// TIA Portal V17 export
// export: Created 2025-03-13T10:31:25.9851877Z, ExportSetting WithDefaults, DisplayName Totally Integrated Automation Portal, DisplayVersion V17 Update 8, DisplayName TIA Portal Openness, DisplayVersion V17 Update 8, DisplayName TIA Portal Version Control Interface, DisplayVersion V17, DisplayName SINAMICS Startdrive Advanced, DisplayVersion V17 SP2, DisplayName SINAMICS Startdrive G110M, G120, G120C, G120D, G120P, G115D, DisplayVersion V17 SP2, DisplayName SINAMICS Startdrive G130, G150, S120, S150, SINAMICS MV, S210, DisplayVersion V17 SP2, DisplayName STEP 7 Professional, DisplayVersion V17 Update 8, DisplayName SINUMERIK ONE STEP 7 Toolbox, DisplayVersion V17 Update 12, DisplayName SINUMERIK 840D sl STEP 7 Toolbox, DisplayVersion V17 Update 12, DisplayName STEP 7 Safety, DisplayVersion V17 Update 6, DisplayName WinCC Advanced, DisplayVersion V17 Update 8
TYPE "FULL_DEPTH_CLADDING"
// stored: IsFailsafeCompliant false
   STRUCT
      FULL_DEPTH : Bool;   // FULL DEPTH / TOTAL FULL DEPTH
      FULL_DEPTH_STA_1 : Bool;   // FULL DEPTH 1 / FULL DEPTH STATION 1
      FULL_DEPTH_STA_2 : Bool;   // FULL DEPTH 2 / FULL DEPTH STATION 2
      FULL_DEPTH_STA_3 : Bool;   // FULL DEPTH 3 / FULL DEPTH STATION 3
      FULL_DEPTH_STA_4 : Bool;   // FULL DEPTH 4 / FULL DEPTH STATION 4
      FULL_DEPTH_STA_5 : Bool;   // FULL DEPTH 5 / FULL DEPTH STATION 5
      FULL_DEPTH_STA_6 : Bool;   // FULL DEPTH 6 / FULL DEPTH STATION 6
      FULL_DEPTH_STA_7 : Bool;   // FULL DEPTH 7 / FULL DEPTH STATION 7
      PART_REJECTED_FIXTURE : Bool;   // PART REJECTED FIXTURE 1 / PART REJECTED FIXTURE
      AUX_FULL_DEPTH_STA_1 : Bool;   // AUXILIARY FULL DEPTH 1 / AUXILIARY FULL DEPTH STATION 1
      AUX_FULL_DEPTH_STA_2 : Bool;   // AUXILIARY FULL DEPTH 2 / AUXILIARY FULL DEPTH STATION 2
      AUX_FULL_DEPTH_STA_3 : Bool;   // AUXILIARY FULL DEPTH 3 / AUXILIARY FULL DEPTH STATION 3
      AUX_FULL_DEPTH_STA_4 : Bool;   // AUXILIARY FULL DEPTH 4 / AUXILIARY FULL DEPTH STATION 4
      AUX_FULL_DEPTH_STA_5 : Bool;   // AUXILIARY FULL DEPTH 5 / AUXILIARY FULL DEPTH STATION 5
      AUX_FULL_DEPTH_STA_6 : Bool;   // AUXILIARY FULL DEPTH 6 / AUXILIARY FULL DEPTH STATION 6
      AUX_FULL_DEPTH_STA_7 : Bool;   // AUXILIARY FULL DEPTH 7 / AUXILIARY FULL DEPTH STATION 7
      AUX_FULL_DEPTH_STA_8 : Bool;   // AUXILIARY FULL DEPTH 8 / AUXILIARY FULL DEPTH STATION 8
      AUX_FULL_DEPTH_PULSE_STA_1 : Bool;   // AUXILIARY FULL DEPTH PULSE 1 / AUXILIARY FULL DEPTH PULSE STATION 1
      AUX_FULL_DEPTH_PULSE_STA_2 : Bool;   // AUXILIARY FULL DEPTH PULSE 2 / AUXILIARY FULL DEPTH PULSE STATION 2
      AUX_FULL_DEPTH_PULSE_STA_3 : Bool;   // AUXILIARY FULL DEPTH PULSE 3 / AUXILIARY FULL DEPTH PULSE STATION 3
      AUX_FULL_DEPTH_PULSE_STA_4 : Bool;   // AUXILIARY FULL DEPTH PULSE 4 / AUXILIARY FULL DEPTH PULSE STATION 4
      AUX_FULL_DEPTH_PULSE_STA_5 : Bool;   // AUXILIARY FULL DEPTH PULSE 5 / AUXILIARY FULL DEPTH PULSE STATION 5
      AUX_FULL_DEPTH_PULSE_STA_6 : Bool;   // AUXILIARY FULL DEPTH PULSE 6 / AUXILIARY FULL DEPTH PULSE STATION 6
      AUX_FULL_DEPTH_PULSE_STA_7 : Bool;   // AUXILIARY FULL DEPTH PULSE 7 / AUXILIARY FULL DEPTH PULSE STATION 7
      AUX_FULL_DEPTH_PULSE_STA_8 : Bool;   // AUXILIARY FULL DEPTH PULSE 8 / AUXILIARY FULL DEPTH PULSE STATION 8
      FD_PULSE : Bool;   // FULL DEPTH PULSE / TOTAL FULL DEPTH PULSE
      FD_STA_1_PULSE : Bool;   // FULL DEPTH 1 PULSE / FULL DEPTH STATION 1 PULSE
      FD_STA_2_PULSE : Bool;   // FULL DEPTH 2 PULSE / FULL DEPTH STATION 2 PULSE
      FD_STA_3_PULSE : Bool;   // FULL DEPTH 3 PULSE / FULL DEPTH STATION 3 PULSE
      FD_STA_4_PULSE : Bool;   // FULL DEPTH 4 PULSE / FULL DEPTH STATION 4 PULSE
      FD_STA_5_PULSE : Bool;   // FULL DEPTH 5 PULSE / FULL DEPTH STATION 5 PULSE
      FD_STA_6_PULSE : Bool;   // FULL DEPTH 6 PULSE / FULL DEPTH STATION 6 PULSE
      FD_STA_7_PULSE : Bool;   // FULL DEPTH 7 PULSE / FULL DEPTH STATION 7 PULSE
   END_STRUCT;
END_TYPE
